FUNCTION_BLOCK Switch IMPLEMENTS ITF_Cylinder
VAR_INPUT
END_VAR
VAR_OUTPUT
END_VAR
VAR
	//Hardware
	DI_Extended AT %I* : BOOL;
	DI_Retracted AT %I* : BOOL;
	DO_Extend AT %Q* : BOOL;
	//NOT USED BUT USABLE
	DI_BoundaryPressure AT %I* : BOOL;
END_VAR

PROPERTY Extended : BOOL
GET
Extended := DI_Extended;
END_GET
END_PROPERTY

METHOD METH_Extend : BOOL
DO_Extend := TRUE;
END_METHOD

METHOD METH_Retract : BOOL
DO_Extend := FALSE;
END_METHOD

PROPERTY Retracted : BOOL
GET
Retracted := DI_Retracted;
END_GET
END_PROPERTY

END_FUNCTION_BLOCK

(* stored: Version 1.1.0.1, ProductVersion 3.1.4024.9
   POU Switch: Id {08aab6e2-fe00-4610-8c46-d809e8a3f02f}, SpecialFunc None
   Property Extended: Id {78489254-2d20-44df-ae19-12644a7ac9b6}
   Get Get: Id {22ac8942-a0de-4d74-9e91-0ed34491a299}
   Method METH_Extend: Id {1c49a489-3b4b-44a9-a37e-d330a129e658}
   Method METH_Retract: Id {93f57fb9-d058-4ec2-8347-ea76a1193289}
   Property Retracted: Id {30f93018-ade1-4d1c-9f06-9efa80dce803}
   Get Get: Id {af4f16b4-19bb-4745-b8d9-8515301a2dd1} *)
